FUNCTION derivcvar_M_Distributing_t : LREAL
VAR_INPUT
	state: STATE;
END_VAR

derivcvar_M_Distributing_t := ifExprFunc1(state);

END_FUNCTION

(* stored: Version 1.1.0.1, ProductVersion 3.1.4022.18
   POU derivcvar_M_Distributing_t: Id {42f1a725-9a71-481c-a9a0-296a175d620e}, SpecialFunc None *)
